{attribute addProperty BoxType "EL5001-0011-0019"}
{attribute addProperty Id "StatusAT %I*Status_EA2B79591621Counter_valueAT %I*UDINT32417"}
{attribute addProperty CRC "2154399983"}
{attribute addProperty SizeInBites "48"}
{attribute addProperty SizeInBytes "6"}
TYPE SSI_Inputs_806988EF :
STRUCT
	{attribute addProperty Name "Status"}
	Status AT %I* : Status_EA2B7959;
	{attribute addProperty Name "Counter_value"}
	Counter_value AT %I* : UDINT;
END_STRUCT
END_TYPE

(* stored: Version 1.2.0.0, ProductVersion 3.1.4024.9
   DUT SSI_Inputs_806988EF: Id {db43eb1b-39b0-414e-a1dc-1caa78f49e03} *)
